(******************************************************************************)
(*	Gate request															  *)
(******************************************************************************)
FUNCTION_BLOCK GateRequest
VAR_INPUT
	GateClosed 			: BOOL; (* Gate closed signal(s) from safety program *)
	SafeState			: BOOL; (* Machine is in safe state *)
	Request_Open 		: BOOL; (* Request door open *)
	Reset				: BOOL; (* Reset Button from safety program *)
	TimeOutSafeState	: TIME:= T#5S; (* Max time for safe state *)
END_VAR
VAR_OUTPUT
	Lock 				: BOOL; (* Activate lock(s) *)
	GateRequest_Light 	: BOOL; (* Light request button *)
	ResetButton_Light 	: BOOL; (* Light reset button *)
END_VAR
VAR
	TimerFlashOn		: TON; (* Timer for flash on *)
	TimerFlashOff		: TON; (* Timer for Flash off *)
	Flash				: SR; (* Flash function *)
END_VAR

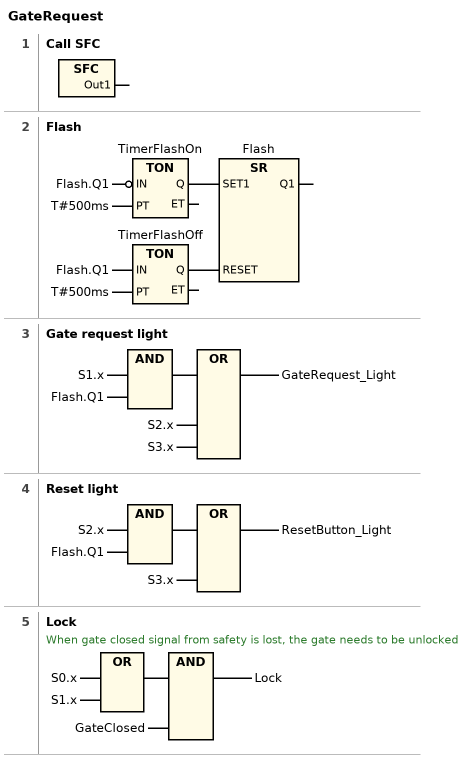
// NETWORK 1: Call SFC
SFC();

// NETWORK 2: Flash
TimerFlashOn(IN := NOT Flash.Q1, PT := T#500ms); // TON
TimerFlashOff(IN := Flash.Q1, PT := T#500ms); // TON
Flash(SET1 := TimerFlashOn.Q, RESET := TimerFlashOff.Q); // SR

// NETWORK 3: Gate request light
GateRequest_Light := S1.x AND Flash.Q1 OR S2.x OR S3.x;

// NETWORK 4: Reset light
ResetButton_Light := S2.x AND Flash.Q1 OR S3.x;

// NETWORK 5: Lock
// When gate closed signal from safety is lost, the gate needs to be unlocked
Lock := (S0.x OR S1.x) AND GateClosed;

ACTION SFC:
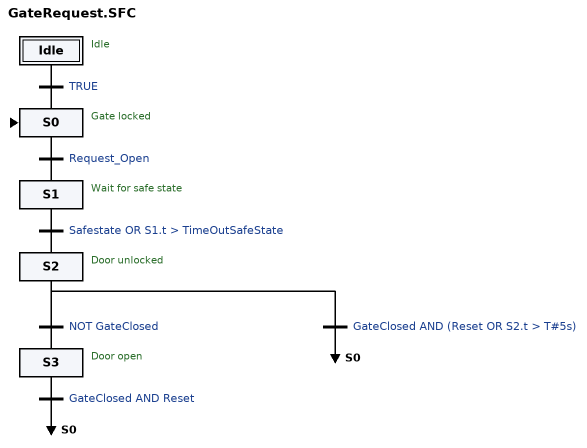
// Idle
INITIAL_STEP Idle:
END_STEP
TRANSITION FROM Idle TO S0
    := TRUE;
END_TRANSITION
// Gate locked
STEP S0:
END_STEP
TRANSITION FROM S0 TO S1
    := Request_Open;
END_TRANSITION
// Wait for safe state
STEP S1:
END_STEP
TRANSITION FROM S1 TO S2
    := Safestate OR S1.t > TimeOutSafeState;
END_TRANSITION
// Door unlocked
STEP S2:
END_STEP
TRANSITION FROM S2 TO S3
    := NOT GateClosed;
END_TRANSITION
TRANSITION FROM S2 TO S0
    := GateClosed AND (Reset OR S2.t > T#5s);
END_TRANSITION
// Door open
STEP S3:
END_STEP
TRANSITION FROM S3 TO S0
    := GateClosed AND Reset;
END_TRANSITION
END_ACTION

END_FUNCTION_BLOCK

(* stored: Version 1.1.0.1, ProductVersion 3.1.4020.12
   POU GateRequest: Id {f5fcf1a6-56f5-427b-9622-9c57f702d2e5}, SpecialFunc None
   Action SFC: Id {77271035-f605-4a7e-b496-77d6ecd0874f} *)
